FUNCTION_BLOCK TRisingEdge
VAR
    R_TRIG1 : R_TRIG;
END_VAR

PROPERTY EdgeDetected : BOOL
GET
EdgeDetected := R_TRIG1.Q;
END_GET
END_PROPERTY

METHOD Test : BOOL
VAR_INPUT
    Value : BOOL;
END_VAR
R_TRIG1(CLK := Value);
Test := R_TRIG1.Q;
END_METHOD

END_FUNCTION_BLOCK

(* stored: Version 1.1.0.1, ProductVersion 3.1.4024.3
   POU TRisingEdge: Id {f6757e14-997b-4fa3-adf7-d19673279582}, SpecialFunc None
   Property EdgeDetected: Id {69ab78d3-83d3-4361-9f6d-953ebd99c416}
   Get Get: Id {3a26e92a-2b1f-4295-82c5-22174ccfa62d}
   Method Test: Id {2bf4e7cb-5fd5-4ce5-afba-102bd83c2305} *)
